  rq_init_comm_if_connected(9, "1")
  rq_init_comm_if_connected(2, "2")
  rq_init_comm_if_connected(3, "3")
  rq_init_comm_if_connected(4, "4")
  rq_print_connected_grippers()
  rq_gripper_communication_thread = run rq_gripper_communication()
  set_closed_norm(100.0, 1)
  set_open_norm(0.0, 1)
  set_closed_mm(0.0, 1)
  set_open_mm(50.0, 1)
  set_closed_norm(100.0, 2)
  set_open_norm(0.0, 2)
  set_closed_mm(0.0, 2)
  set_open_mm(50.0, 2)
  set_closed_norm(100.0, 3)
  set_open_norm(0.0, 3)
  set_closed_mm(0.0, 3)
  set_open_mm(50.0, 3)
  set_closed_norm(100.0, 4)
  set_open_norm(0.0, 4)
  set_closed_mm(0.0, 4)
  set_open_mm(50.0, 4)
  rq_current_limit_enabled = False
  while(not rq_gripper_communication_thread_started):
      sleep(0.008)
  end
  # end: URCap Installation Node
  global Pallet_2_cnt_3=1
  global Pallet_2_cnt_4=1
  global Pallet_2_cnt_5=1
  global Pallet_2_cnt_6=1
  global Pallet_2_lct_3=1
  global Pallet_2_lct_4=1
  global Pallet_2_lct_5=1
  global Pallet_2_lct_6=1
  global Pallet_2_lno_3=1
  global Pallet_2_lno_4=1
  global Pallet_2_lno_5=1
  global Pallet_2_lno_6=1
  global Pallet_2_sep_3= False
  global Pallet_2_sep_4= False
  global Pallet_2_sep_5= False
  global Pallet_2_sep_6= False
  global Pallet_2_tct_3=1
  global Pallet_2_tct_4=1
  global Pallet_2_tct_5=1
  global Pallet_2_tct_6=1
  global qNearApproach=[0,0,0,0,0,0]
  global qNearApproach_1=[0,0,0,0,0,0]
  global qNearApproach_2=[0,0,0,0,0,0]
  global qNearApproach_3=[0,0,0,0,0,0]
  global Waypoint_2_p=p[.497545315671, .066443275206, .565567908320, 2.166165135185, -2.096986285032, -.058830025629]
  global Waypoint_2_q=[3.020538828963275, -1.5350072347942687, 1.310240075700583, -1.2376589337904829, -1.6454681359193124, -0.14796686856282548]
  global Approach_1_p=p[.529811548736, .078794296821, -.249075713058, 2.252782682541, -2.172328817817, .036580928376]
  global Approach_1_q=[3.039864276185085, -0.18566656279727667, 1.7536743022026577, -3.1489013797878584, -1.5954024336410413, -0.13295549283606078]
  global ToolActionPoi_1_p=p[.529805653595, .078793026024, -.279911555553, 2.252768683998, -2.172326347106, .036578768693]
  global ToolActionPoi_1_q=[3.039744912416083, -0.11220692465133553, 1.6920841553070907, -3.16078404588802, -1.5955704096675678, -0.13312653598666024]
  global Exit_2_p=p[.529810238319, .078794594586, -.211983202439, 2.252768831616, -2.172321661670, .036580192861]
  global Exit_2_q=[3.0400074576796485, -0.2750556215204334, 1.820883845919285, -3.1267173172014413, -1.5952202467689496, -0.13278613781927362]
  global Approach_p=p[.259939147756, -.683221746138, .330823595725, .096711987287, 3.097647085282, .045794034220]
  global Approach_q=[1.7433785897016765, -0.9789911612274125, 1.1929114404367116, -1.7636157466916895, -1.5217364879006539, 0.23748448608004402]
  global ToolActionPoint_p=p[.260951127880, -.682556749615, .307415310056, .096720171615, 3.097650623093, .045741938859]
  global ToolActionPoint_q=[1.7448971700273574, -0.9655793386006408, 1.2326464916352902, -1.816818537032935, -1.5217211095327015, 0.23910702792430083]
  global Exit_1_p=p[.258824165549, -.683958688734, .356887144820, .096737432605, 3.097619259377, .045729561599]
  global Exit_1_q=[1.741693917054314, -0.990422118385399, 1.1437541193824776, -1.7029416535283248, -1.5217729231978865, 0.23566896849839264]
  while (True):
    $ 2 "Robot Program"
    $ 3 "Home (Safe)"
    movej([2.5829941725145966, -1.8029425748621035, 2.4397996453919744, -3.810050312281298, -1.0067438250200702, 0.02806297247002032], a=1.3962634015954636, v=1.0471975511965976)
    # begin: URCap Program Node
    #   Source: EnabledRobotics - ER-ABILITY, 5.0.0, Enabled Robotics ApS
    #   Type: ER-Ability
    $ 4 "ER-Ability"
    __er_thread_handle = 0
    daemon=rpc_factory("xmlrpc", "http://192.168.11.40:4568")
    daemon.set_init_status(0)
    HOST_IP = ""
    interpreter_mode(clearQueueOnEnter=False, clearOnEnd=False)
    if (not daemon.connect(HOST_IP)):
      textmsg("Failed to connect to ability")
      halt
    end
    thread __er_connection_watchdog():
      while (True):
        if (not daemon.watchdog()):
          textmsg("Lost connection to ability")
          halt
        end
        sleep(3.0)
      end
    end
    def sendError(errorMsg):
    daemon.send_error(errorMsg)
  end
  daemon.set_init_status(1)
  __er_watchdog_handle = run __er_connection_watchdog()
  interpreter_mode(clearQueueOnEnter=False, clearOnEnd=False)
  # begin: URCap Program Node
  #   Source: EnabledRobotics - ER-ABILITY, 5.0.0, Enabled Robotics ApS
  #   Type: EventNode
  $ 5 "EventNode: GripOpen" "noBreak"
  def GripOpen_definition():
  # begin: URCap Program Node
  #   Source: Robotiq_Grippers, 2.4.0.45103, Robotiq Inc.
  #   Type: Gripper
  $ 6 "Gripper Open (1)" "noBreak"
  if not(gripper_connected[0]):
    popup("Gripper 1 must be connected to run this program.", "No connection", False, True, True)
  end
  if not(rq_is_gripper_activated("1")):
    popup("Gripper 1 is not activated. Go to Installation tab > Gripper to activate it and run the program again.", "Not activated", False, True, True)
  end
  rq_set_pos_spd_for(0, 255, 255, "1")
  rq_wait_pos_spe_for_request(0, 255, 255, "1")
  rq_go_to("1")
  rq_wait("1")
  # end: URCap Program Node
  end
  thread GripOpen_thread():
  GripOpen_definition()
  daemon.done_executing()
  end
  def GripOpen():
  textmsg("Executing event: GripOpen")
  __er_thread_handle = run GripOpen_thread()
  end
  if (not daemon.register_method("GripOpen","[]", False)):
    textmsg("Failed to connect to register method GripOpen")
    halt
  end
  sync()
  # end: URCap Program Node
  # begin: URCap Program Node
  #   Source: EnabledRobotics - ER-ABILITY, 5.0.0, Enabled Robotics ApS
  #   Type: EventNode
  $ 7 "EventNode: GripClosed" "noBreak"
  def GripClosed_definition():
  # begin: URCap Program Node
  #   Source: Robotiq_Grippers, 2.4.0.45103, Robotiq Inc.
  #   Type: Gripper
  $ 8 "Gripper Close (1)" "noBreak"
  if not(gripper_connected[0]):
    popup("Gripper 1 must be connected to run this program.", "No connection", False, True, True)
  end
  if not(rq_is_gripper_activated("1")):
    popup("Gripper 1 is not activated. Go to Installation tab > Gripper to activate it and run the program again.", "Not activated", False, True, True)
  end
  rq_set_pos_spd_for(255, 255, 179, "1")
  rq_wait_pos_spe_for_request(255, 255, 179, "1")
  rq_go_to("1")
  rq_wait("1")
  # end: URCap Program Node
  end
  thread GripClosed_thread():
  GripClosed_definition()
  daemon.done_executing()
  end
  def GripClosed():
  textmsg("Executing event: GripClosed")
  __er_thread_handle = run GripClosed_thread()
  end
  if (not daemon.register_method("GripClosed","[]", False)):
    textmsg("Failed to connect to register method GripClosed")
    halt
  end
  sync()
  # end: URCap Program Node
  # begin: URCap Program Node
  #   Source: EnabledRobotics - ER-ABILITY, 5.0.0, Enabled Robotics ApS
  #   Type: EventNode
  $ 9 "EventNode: Unload" "noBreak"
  global __er_Unload_arg_pose = p[0, 0, 0, 0, 0, 0]
  def Unload_definition(arg_pose):
  $ 10 "Unload_ref≔__er_Unload_arg_pose" "noBreak"
  global Unload_ref=__er_Unload_arg_pose
  $ 11 "MoveJ" "noBreak"
  $ 12 "Waypoint_2" "noBreak"
  movej(get_inverse_kin(Waypoint_2_p, qnear=Waypoint_2_q), a=1.3962634015954636, v=1.0471975511965976)
  $ 13 "Pallet_5" "noBreak"
  def Pallet_5_trans(pose):
  return p[pose[0], pose[1], pose[2], 0, 0, 0]
  end
  def Pallet_5_rot(pose):
  return p[0, 0, 0, pose[3], pose[4], pose[5]]
  end
  def Pallet_5_compute_pallet_waypoint(T_base_feature_taught, T_feature_referencePoint_taught, T_referencePoint_approach_taught, T_base_feature, T_base_referencePoint):
  local trans_referencePoint_approach_in_feature_taught = pose_sub(Pallet_5_trans(pose_trans(T_feature_referencePoint_taught, T_referencePoint_approach_taught)), Pallet_5_trans(T_feature_referencePoint_taught))
  local rot_referencePoint_approach_in_feature_taught = pose_trans(Pallet_5_rot(T_feature_referencePoint_taught), pose_trans(Pallet_5_rot(T_referencePoint_approach_taught), pose_inv(Pallet_5_rot(T_feature_referencePoint_taught))))
  T_feature_referencePoint = pose_trans(pose_inv(T_base_feature), T_base_referencePoint)
  rot_referencePoint_approach = pose_trans(pose_inv(Pallet_5_rot(T_feature_referencePoint)), pose_trans(rot_referencePoint_approach_in_feature_taught, Pallet_5_rot(T_feature_referencePoint)))
  T_feature_approach = pose_trans(trans_referencePoint_approach_in_feature_taught, pose_trans(T_feature_referencePoint, rot_referencePoint_approach))
  T_base_approach = pose_trans(T_base_feature, T_feature_approach)
  return T_base_approach
  end
  Pallet_2_tct_6 = 3
  if (Pallet_2_cnt_6 > 3 or Pallet_2_cnt_6 < 1):
    Pallet_2_cnt_6 = 1
  end
  $ 14 "Patterns" "noBreak"
  $ 15 "Line_Pattern_7" "noBreak"
  $ 18 "Layers" "noBreak"
  if (Pallet_2_cnt_6 < 4):
    Pallet_2_lno_6 = 1
    Pallet_2_lct_6 = Pallet_2_cnt_6
    global StartItem_7=pose_trans(p[0.0,0.0,0.0,0.0,0.0,0.0], pose_trans(p[-.000000000000, -.000000000000, -.000000000000, .000000000000, .000000000000, .000000000000], p[.529805653595, .078793026024, -.279911555553, 2.252768683999, -2.172326347101, .036578768700]))
    global EndItem_7=pose_trans(p[0.0,0.0,0.0,0.0,0.0,0.0], pose_trans(p[-.000000000000, -.000000000000, -.000000000000, .000000000000, .000000000000, .000000000000], p[.533401069223, -.101391020004, -.279793718806, 2.252783599118, -2.172333887579, .036654201565]))
    referencePoin_1 = interpolate_pose(StartItem_7, EndItem_7, (Pallet_2_lct_6 - 1)/2)
    if ((Pallet_2_lct_6 - 1) < 1.5):
      qNearApproach_1 = [2.885448189355559, 0.43603101886187573, 1.512248322517327, -5.09598803422031, -1.2812075252986297, -0.023929430846770572]
    else:
      qNearApproach_1 = [2.272042773983432, 0.4199865702204392, 1.4836778687882308, -5.05440269585694, -0.667839702259915, -0.018231839794984772]
    end
    direction = p[0,0,1,0,0,0]
    referencePoin_1 = pose_add (referencePoin_1,p[0.0*direction[0],0.0*direction[1],0.0*direction[2],0,0,0])
  end
  Approach_1_p = Pallet_5_compute_pallet_waypoint(p[0.0,0.0,0.0,0.0,0.0,0.0], pose_trans(pose_inv(p[0.0,0.0,0.0,0.0,0.0,0.0]), p[0.5298056535954119,0.07879302602441744,-0.279911555552729,2.2527686839987453,-2.1723263471008782,0.03657876870047535]), p[7.713003808866858E-4,-2.4326214461312112E-4,-0.030825235408129148,9.465437041250408E-6,-7.291023033565463E-6,-4.926570927565642E-6], p[0.0,0.0,0.0,0.0,0.0,0.0], referencePoin_1)
  Approach_1_p = pose_trans(p[0.5298056535954119,0.07879302602441744,-0.279911555552729,2.252768683998824,-2.1723263471009577,0.03657876870045813], pose_trans(pose_inv(referencePoin_1), Approach_1_p))
  Approach_1_q = qNearApproach_1
  ToolActionPoi_1_p = Pallet_5_compute_pallet_waypoint(p[0.0,0.0,0.0,0.0,0.0,0.0], pose_trans(pose_inv(p[0.0,0.0,0.0,0.0,0.0,0.0]), p[0.5298056535954119,0.07879302602441744,-0.279911555552729,2.2527686839987453,-2.1723263471008782,0.03657876870047535]), p[1.3877787807814457E-17,0.0,0.0,0.0,0.0,0.0], p[0.0,0.0,0.0,0.0,0.0,0.0], referencePoin_1)
  ToolActionPoi_1_p = pose_trans(p[0.5298056535954119,0.07879302602441744,-0.279911555552729,2.252768683998824,-2.1723263471009577,0.03657876870045813], pose_trans(pose_inv(referencePoin_1), ToolActionPoi_1_p))
  Exit_2_p = Pallet_5_compute_pallet_waypoint(p[0.0,0.0,0.0,0.0,0.0,0.0], pose_trans(pose_inv(p[0.0,0.0,0.0,0.0,0.0,0.0]), p[0.5298056535954119,0.07879302602441744,-0.279911555552729,2.2527686839987453,-2.1723263471008782,0.03657876870047535]), p[0.0017000247291813209,-5.274420544957303E-4,-0.06790502854043742,-1.5766278052156214E-6,2.8353740061571936E-6,-2.251562946520516E-6], p[0.0,0.0,0.0,0.0,0.0,0.0], referencePoin_1)
  Exit_2_p = pose_trans(p[0.5298056535954119,0.07879302602441744,-0.279911555552729,2.252768683998824,-2.1723263471009577,0.03657876870045813], pose_trans(pose_inv(referencePoin_1), Exit_2_p))
  $ 19 "At Each Item" "noBreak"
  $ 20 "Generated Movements" "noBreak"
  $ 21 "MoveJ" "noBreak"
  $ 22 "Approach_1" "noBreak"
  movej(get_inverse_kin(pose_trans(referencePoin_1, pose_trans(p[.066528706245, .530155020651, -.282422442075, -2.252768683999, 2.172326347101, -.036578768700], Approach_1_p)), qnear=Approach_1_q), a=1.3962634015954636, v=1.0471975511965976)
  $ 23 "MoveL" "noBreak"
  $ 24 "ToolActionPoi_1" "noBreak"
  movel(pose_trans(referencePoin_1, pose_trans(p[.066528706245, .530155020651, -.282422442075, -2.252768683999, 2.172326347101, -.036578768700], ToolActionPoi_1_p)), a=1.2, v=0.25)
  $ 25 "Tool action" "noBreak"
  # begin: URCap Program Node
  #   Source: Robotiq_Grippers, 2.4.0.45103, Robotiq Inc.
  #   Type: Gripper
  $ 26 "Gripper Close (1)" "noBreak"
  if not(gripper_connected[0]):
    popup("Gripper 1 must be connected to run this program.", "No connection", False, True, True)
  end
  if not(rq_is_gripper_activated("1")):
    popup("Gripper 1 is not activated. Go to Installation tab > Gripper to activate it and run the program again.", "Not activated", False, True, True)
  end
  rq_set_pos_spd_for(255, 255, 255, "1")
  rq_wait_pos_spe_for_request(255, 255, 255, "1")
  rq_go_to("1")
  rq_wait("1")
  # end: URCap Program Node
  $ 27 "MoveL" "noBreak"
  $ 28 "Exit_2" "noBreak"
  movel(pose_trans(referencePoin_1, pose_trans(p[.066528706245, .530155020651, -.282422442075, -2.252768683999, 2.172326347101, -.036578768700], Exit_2_p)), a=1.2, v=0.25)
  Pallet_2_sep_6 = False
  if (Pallet_2_cnt_6 >= 3):
    Pallet_2_cnt_6 = 1
  else:
    Pallet_2_cnt_6 = Pallet_2_cnt_6 + 1
  end
  $ 29 "MoveJ" "noBreak"
  $ 30 "Waypoint_2" "noBreak"
  movej(get_inverse_kin(Waypoint_2_p, qnear=Waypoint_2_q), a=1.3962634015954636, v=1.0471975511965976)
  $ 31 "Pallet_1" "noBreak"
  def Pallet_1_trans(pose):
  return p[pose[0], pose[1], pose[2], 0, 0, 0]
  end
  def Pallet_1_rot(pose):
  return p[0, 0, 0, pose[3], pose[4], pose[5]]
  end
  def Pallet_1_compute_pallet_waypoint(T_base_feature_taught, T_feature_referencePoint_taught, T_referencePoint_approach_taught, T_base_feature, T_base_referencePoint):
  local trans_referencePoint_approach_in_feature_taught = pose_sub(Pallet_1_trans(pose_trans(T_feature_referencePoint_taught, T_referencePoint_approach_taught)), Pallet_1_trans(T_feature_referencePoint_taught))
  local rot_referencePoint_approach_in_feature_taught = pose_trans(Pallet_1_rot(T_feature_referencePoint_taught), pose_trans(Pallet_1_rot(T_referencePoint_approach_taught), pose_inv(Pallet_1_rot(T_feature_referencePoint_taught))))
  T_feature_referencePoint = pose_trans(pose_inv(T_base_feature), T_base_referencePoint)
  rot_referencePoint_approach = pose_trans(pose_inv(Pallet_1_rot(T_feature_referencePoint)), pose_trans(rot_referencePoint_approach_in_feature_taught, Pallet_1_rot(T_feature_referencePoint)))
  T_feature_approach = pose_trans(trans_referencePoint_approach_in_feature_taught, pose_trans(T_feature_referencePoint, rot_referencePoint_approach))
  T_base_approach = pose_trans(T_base_feature, T_feature_approach)
  return T_base_approach
  end
  Pallet_2_tct_5 = 3
  if (Pallet_2_cnt_5 > 3 or Pallet_2_cnt_5 < 1):
    Pallet_2_cnt_5 = 1
  end
  $ 32 "Patterns" "noBreak"
  $ 33 "Line_Pattern_1" "noBreak"
  $ 36 "Layers" "noBreak"
  if (Pallet_2_cnt_5 < 4):
    Pallet_2_lno_5 = 1
    Pallet_2_lct_5 = Pallet_2_cnt_5
    global StartItem_1=pose_trans(Unload_ref, pose_trans(p[.418279672309, .619551005398, .340218691369, -.096685752657, -3.097655012832, -.045744274097], p[.260951127880, -.682556749615, .307415310056, .096720171636, 3.097650623082, .045741938829]))
    global EndItem_1=pose_trans(Unload_ref, pose_trans(p[.418279672309, .619551005398, .340218691369, -.096685752657, -3.097655012832, -.045744274097], p[.082322324479, -.670818754149, .307468197109, .096703817876, 3.097665036034, .045785718306]))
    referencePoin_2 = interpolate_pose(StartItem_1, EndItem_1, (Pallet_2_lct_5 - 1)/2)
    if ((Pallet_2_lct_5 - 1) < 1.5):
      qNearApproach_2 = [3.3641552695356225, -0.8479015660023324, 1.98966712800588, -1.131219804936615, -2.916013250302344, 0.010451340576699941]
    else:
      qNearApproach_2 = [3.300396662600974, -0.612779437790441, 1.4440990949301122, -0.8163897168853449, -2.98016670938038, 0.01484693428962075]
    end
    direction = pose_trans(p[0,0,0,Unload_ref[3],Unload_ref[4],Unload_ref[5]], p[0,0,1,0,0,0])
    referencePoin_2 = pose_add (referencePoin_2,p[0.0*direction[0],0.0*direction[1],0.0*direction[2],0,0,0])
  end
  Approach_p = Pallet_1_compute_pallet_waypoint(p[0.3642472151847146,-0.6539896130686794,0.3378929456834839,0.09668575265698816,3.0976550128318143,0.04574427409651193], pose_trans(pose_inv(p[0.3642472151847146,-0.6539896130686794,0.3378929456834839,0.09668575265698816,3.0976550128318143,0.04574427409651193]), p[0.260951127880279,-0.6825567496145907,0.307415310056378,0.09672017163594536,3.0976506230824565,0.04574193882899084]), p[4.300908552967719E-6,-4.9422491205097785E-6,-0.023439584449423678,-3.3818317637974754E-5,-1.900639287119668E-6,-4.541078724455231E-6], Unload_ref, referencePoin_2)
  Approach_p = pose_trans(p[0.2609511278802791,-0.6825567496145908,0.30741531005637773,0.0967201716359448,3.0976506230824357,0.04574193882899086], pose_trans(pose_inv(referencePoin_2), Approach_p))
  Approach_q = qNearApproach_2
  ToolActionPoint_p = Pallet_1_compute_pallet_waypoint(p[0.3642472151847146,-0.6539896130686794,0.3378929456834839,0.09668575265698816,3.0976550128318143,0.04574427409651193], pose_trans(pose_inv(p[0.3642472151847146,-0.6539896130686794,0.3378929456834839,0.09668575265698816,3.0976550128318143,0.04574427409651193]), p[0.260951127880279,-0.6825567496145907,0.307415310056378,0.09672017163594536,3.0976506230824565,0.04574193882899084]), p[5.551115123125783E-17,1.1102230246251565E-16,-3.3306690738754696E-16,0.0,0.0,0.0], Unload_ref, referencePoin_2)
  ToolActionPoint_p = pose_trans(p[0.2609511278802791,-0.6825567496145908,0.30741531005637773,0.0967201716359448,3.0976506230824357,0.04574193882899086], pose_trans(pose_inv(referencePoin_2), ToolActionPoint_p))
  Exit_1_p = Pallet_1_compute_pallet_waypoint(p[0.3642472151847146,-0.6539896130686794,0.3378929456834839,0.09668575265698816,3.0976550128318143,0.04574427409651193], pose_trans(pose_inv(p[0.3642472151847146,-0.6539896130686794,0.3378929456834839,0.09668575265698816,3.0976550128318143,0.04574427409651193]), p[0.260951127880279,-0.6825567496145907,0.307415310056378,0.09672017163594536,3.0976506230824565,0.04574193882899084]), p[-2.4468940774680092E-6,-6.239484140468932E-6,-0.04953737772677924,6.96031944656997E-6,-3.138925438944591E-5,1.1138535086107724E-5], Unload_ref, referencePoin_2)
  Exit_1_p = pose_trans(p[0.2609511278802791,-0.6825567496145908,0.30741531005637773,0.0967201716359448,3.0976506230824357,0.04574193882899086], pose_trans(pose_inv(referencePoin_2), Exit_1_p))
  $ 37 "At Each Item" "noBreak"
  $ 38 "Generated Movements" "noBreak"
  $ 39 "MoveJ" "noBreak"
  $ 40 "Approach" "noBreak"
  movej(get_inverse_kin(pose_trans(referencePoin_2, pose_trans(p[.315836214354, .655355973761, .315022878219, -.096720171636, -3.097650623082, -.045741938829], Approach_p)), qnear=Approach_q), a=1.3962634015954636, v=1.0471975511965976)
  $ 41 "MoveL" "noBreak"
  $ 42 "ToolActionPoint" "noBreak"
  movel(pose_trans(referencePoin_2, pose_trans(p[.315836214354, .655355973761, .315022878219, -.096720171636, -3.097650623082, -.045741938829], ToolActionPoint_p)), a=1.2, v=0.25)
  $ 43 "Tool action" "noBreak"
  # begin: URCap Program Node
  #   Source: Robotiq_Grippers, 2.4.0.45103, Robotiq Inc.
  #   Type: Gripper
  $ 44 "Gripper Open (1)" "noBreak"
  if not(gripper_connected[0]):
    popup("Gripper 1 must be connected to run this program.", "No connection", False, True, True)
  end
  if not(rq_is_gripper_activated("1")):
    popup("Gripper 1 is not activated. Go to Installation tab > Gripper to activate it and run the program again.", "Not activated", False, True, True)
  end
  rq_set_pos_spd_for(0, 255, 255, "1")
  rq_wait_pos_spe_for_request(0, 255, 255, "1")
  rq_go_to("1")
  rq_wait("1")
  # end: URCap Program Node
  $ 45 "MoveL" "noBreak"
  $ 46 "Exit_1" "noBreak"
  movel(pose_trans(referencePoin_2, pose_trans(p[.315836214354, .655355973761, .315022878219, -.096720171636, -3.097650623082, -.045741938829], Exit_1_p)), a=1.2, v=0.25)
  Pallet_2_sep_5 = False
  if (Pallet_2_cnt_5 >= 3):
    Pallet_2_cnt_5 = 1
  else:
    Pallet_2_cnt_5 = Pallet_2_cnt_5 + 1
  end
  $ 47 "MoveJ" "noBreak"
  $ 48 "Waypoint_2" "noBreak"
  movej(get_inverse_kin(Waypoint_2_p, qnear=Waypoint_2_q), a=1.3962634015954636, v=1.0471975511965976)
  end
  thread Unload_thread():
  Unload_definition(__er_Unload_arg_pose)
  daemon.done_executing()
  end
  def Unload(arg_pose):
  textmsg("Executing event: Unload, with arguments:")
  textmsg("Argument: arg_pose = ", arg_pose)
  __er_Unload_arg_pose = arg_pose
  __er_thread_handle = run Unload_thread()
  end
  if (not daemon.register_method("Unload","[pose]", False)):
    textmsg("Failed to connect to register method Unload")
    halt
  end
  sync()
  # end: URCap Program Node
  # begin: URCap Program Node
  #   Source: EnabledRobotics - ER-ABILITY, 5.0.0, Enabled Robotics ApS
  #   Type: EventNode
  $ 49 "EventNode: Palletize" "noBreak"
  global __er_Palletize_arg_pose = p[0, 0, 0, 0, 0, 0]
  def Palletize_definition(arg_pose):
  $ 50 "Pallet_ref≔__er_Palletize_arg_pose" "noBreak"
  global Pallet_ref=__er_Palletize_arg_pose
  $ 51 "MoveJ" "noBreak"
  $ 52 "Waypoint_2" "noBreak"
  movej(get_inverse_kin(Waypoint_2_p, qnear=Waypoint_2_q), a=1.3962634015954636, v=1.0471975511965976)
  $ 53 "Pallet_3" "noBreak"
  def Pallet_3_trans(pose):
  return p[pose[0], pose[1], pose[2], 0, 0, 0]
  end
  def Pallet_3_rot(pose):
  return p[0, 0, 0, pose[3], pose[4], pose[5]]
  end
  def Pallet_3_compute_pallet_waypoint(T_base_feature_taught, T_feature_referencePoint_taught, T_referencePoint_approach_taught, T_base_feature, T_base_referencePoint):
  local trans_referencePoint_approach_in_feature_taught = pose_sub(Pallet_3_trans(pose_trans(T_feature_referencePoint_taught, T_referencePoint_approach_taught)), Pallet_3_trans(T_feature_referencePoint_taught))
  local rot_referencePoint_approach_in_feature_taught = pose_trans(Pallet_3_rot(T_feature_referencePoint_taught), pose_trans(Pallet_3_rot(T_referencePoint_approach_taught), pose_inv(Pallet_3_rot(T_feature_referencePoint_taught))))
  T_feature_referencePoint = pose_trans(pose_inv(T_base_feature), T_base_referencePoint)
  rot_referencePoint_approach = pose_trans(pose_inv(Pallet_3_rot(T_feature_referencePoint)), pose_trans(rot_referencePoint_approach_in_feature_taught, Pallet_3_rot(T_feature_referencePoint)))
  T_feature_approach = pose_trans(trans_referencePoint_approach_in_feature_taught, pose_trans(T_feature_referencePoint, rot_referencePoint_approach))
  T_base_approach = pose_trans(T_base_feature, T_feature_approach)
  return T_base_approach
  end
  Pallet_2_tct_3 = 3
  if (Pallet_2_cnt_3 > 3 or Pallet_2_cnt_3 < 1):
    Pallet_2_cnt_3 = 1
  end
  $ 54 "Patterns" "noBreak"
  $ 55 "Line_Pattern_5" "noBreak"
  $ 58 "Layers" "noBreak"
  if (Pallet_2_cnt_3 < 4):
    Pallet_2_lno_3 = 1
    Pallet_2_lct_3 = Pallet_2_cnt_3
    global StartItem_5=pose_trans(Pallet_ref, pose_trans(p[.418279672309, .619551005398, .340218691369, -.096685752657, -3.097655012832, -.045744274097], p[.260951127880, -.682556749615, .307415310056, .096720171636, 3.097650623082, .045741938829]))
    global EndItem_5=pose_trans(Pallet_ref, pose_trans(p[.418279672309, .619551005398, .340218691369, -.096685752657, -3.097655012832, -.045744274097], p[.082322324479, -.670818754149, .307468197109, .096703817876, 3.097665036034, .045785718306]))
    referencePoin_3 = interpolate_pose(StartItem_5, EndItem_5, (Pallet_2_lct_3 - 1)/2)
    if ((Pallet_2_lct_3 - 1) < 1.5):
      qNearApproach = [1.8853350729711007, -0.9945419025980371, 1.8756705078246672, -3.9864826836818184, -1.9494013418490388, 0.0576506840721043]
    else:
      qNearApproach = [1.4834301388931141, -1.1270563789595887, 2.126921432265375, -4.109054351196034, -1.5477728899200969, 0.04377366676978213]
    end
    direction = pose_trans(p[0,0,0,Pallet_ref[3],Pallet_ref[4],Pallet_ref[5]], p[0,0,1,0,0,0])
    referencePoin_3 = pose_add (referencePoin_3,p[0.0*direction[0],0.0*direction[1],0.0*direction[2],0,0,0])
  end
  Approach_p = Pallet_3_compute_pallet_waypoint(p[0.3642472151847146,-0.6539896130686794,0.3378929456834839,0.09668575265698816,3.0976550128318143,0.04574427409651193], pose_trans(pose_inv(p[0.3642472151847146,-0.6539896130686794,0.3378929456834839,0.09668575265698816,3.0976550128318143,0.04574427409651193]), p[0.260951127880279,-0.6825567496145907,0.307415310056378,0.09672017163594536,3.0976506230824565,0.04574193882899084]), p[4.300908552967719E-6,-4.9422491205097785E-6,-0.023439584449423678,-3.3818317637974754E-5,-1.900639287119668E-6,-4.541078724455231E-6], Pallet_ref, referencePoin_3)
  Approach_p = pose_trans(p[0.2609511278802791,-0.6825567496145908,0.30741531005637773,0.0967201716359448,3.0976506230824357,0.04574193882899086], pose_trans(pose_inv(referencePoin_3), Approach_p))
  Approach_q = qNearApproach
  ToolActionPoint_p = Pallet_3_compute_pallet_waypoint(p[0.3642472151847146,-0.6539896130686794,0.3378929456834839,0.09668575265698816,3.0976550128318143,0.04574427409651193], pose_trans(pose_inv(p[0.3642472151847146,-0.6539896130686794,0.3378929456834839,0.09668575265698816,3.0976550128318143,0.04574427409651193]), p[0.260951127880279,-0.6825567496145907,0.307415310056378,0.09672017163594536,3.0976506230824565,0.04574193882899084]), p[5.551115123125783E-17,1.1102230246251565E-16,-3.3306690738754696E-16,0.0,0.0,0.0], Pallet_ref, referencePoin_3)
  ToolActionPoint_p = pose_trans(p[0.2609511278802791,-0.6825567496145908,0.30741531005637773,0.0967201716359448,3.0976506230824357,0.04574193882899086], pose_trans(pose_inv(referencePoin_3), ToolActionPoint_p))
  Exit_1_p = Pallet_3_compute_pallet_waypoint(p[0.3642472151847146,-0.6539896130686794,0.3378929456834839,0.09668575265698816,3.0976550128318143,0.04574427409651193], pose_trans(pose_inv(p[0.3642472151847146,-0.6539896130686794,0.3378929456834839,0.09668575265698816,3.0976550128318143,0.04574427409651193]), p[0.260951127880279,-0.6825567496145907,0.307415310056378,0.09672017163594536,3.0976506230824565,0.04574193882899084]), p[-2.4468940774680092E-6,-6.239484140468932E-6,-0.04953737772677924,6.96031944656997E-6,-3.138925438944591E-5,1.1138535086107724E-5], Pallet_ref, referencePoin_3)
  Exit_1_p = pose_trans(p[0.2609511278802791,-0.6825567496145908,0.30741531005637773,0.0967201716359448,3.0976506230824357,0.04574193882899086], pose_trans(pose_inv(referencePoin_3), Exit_1_p))
  $ 59 "At Each Item" "noBreak"
  $ 60 "Generated Movements" "noBreak"
  $ 61 "MoveJ" "noBreak"
  $ 62 "Approach" "noBreak"
  set_tcp(p[0.0,0.0,0.0,0.0,0.0,0.0])
  movej(get_inverse_kin(pose_trans(referencePoin_3, pose_trans(p[.315836214354, .655355973761, .315022878219, -.096720171636, -3.097650623082, -.045741938829], Approach_p)), qnear=Approach_q), a=1.3962634015954636, v=1.0471975511965976)
  $ 63 "MoveL" "noBreak"
  $ 64 "ToolActionPoint" "noBreak"
  movel(pose_trans(referencePoin_3, pose_trans(p[.315836214354, .655355973761, .315022878219, -.096720171636, -3.097650623082, -.045741938829], ToolActionPoint_p)), a=1.2, v=0.25)
  $ 65 "Tool action" "noBreak"
  # begin: URCap Program Node
  #   Source: Robotiq_Grippers, 2.4.0.45103, Robotiq Inc.
  #   Type: Gripper
  $ 66 "Gripper Close (1)" "noBreak"
  if not(gripper_connected[0]):
    popup("Gripper 1 must be connected to run this program.", "No connection", False, True, True)
  end
  if not(rq_is_gripper_activated("1")):
    popup("Gripper 1 is not activated. Go to Installation tab > Gripper to activate it and run the program again.", "Not activated", False, True, True)
  end
  rq_set_pos_spd_for(255, 250, 0, "1")
  rq_wait_pos_spe_for_request(255, 250, 0, "1")
  rq_go_to("1")
  rq_wait("1")
  # end: URCap Program Node
  $ 67 "MoveL" "noBreak"
  $ 68 "Exit_1" "noBreak"
  movel(pose_trans(referencePoin_3, pose_trans(p[.315836214354, .655355973761, .315022878219, -.096720171636, -3.097650623082, -.045741938829], Exit_1_p)), a=1.2, v=0.25)
  Pallet_2_sep_3 = False
  if (Pallet_2_cnt_3 >= 3):
    Pallet_2_cnt_3 = 1
  else:
    Pallet_2_cnt_3 = Pallet_2_cnt_3 + 1
  end
  $ 69 "MoveJ" "noBreak"
  $ 70 "Waypoint_2" "noBreak"
  movej(get_inverse_kin(Waypoint_2_p, qnear=Waypoint_2_q), a=1.3962634015954636, v=1.0471975511965976)
  $ 71 "Pallet_4" "noBreak"
  def Pallet_4_trans(pose):
  return p[pose[0], pose[1], pose[2], 0, 0, 0]
  end
  def Pallet_4_rot(pose):
  return p[0, 0, 0, pose[3], pose[4], pose[5]]
  end
  def Pallet_4_compute_pallet_waypoint(T_base_feature_taught, T_feature_referencePoint_taught, T_referencePoint_approach_taught, T_base_feature, T_base_referencePoint):
  local trans_referencePoint_approach_in_feature_taught = pose_sub(Pallet_4_trans(pose_trans(T_feature_referencePoint_taught, T_referencePoint_approach_taught)), Pallet_4_trans(T_feature_referencePoint_taught))
  local rot_referencePoint_approach_in_feature_taught = pose_trans(Pallet_4_rot(T_feature_referencePoint_taught), pose_trans(Pallet_4_rot(T_referencePoint_approach_taught), pose_inv(Pallet_4_rot(T_feature_referencePoint_taught))))
  T_feature_referencePoint = pose_trans(pose_inv(T_base_feature), T_base_referencePoint)
  rot_referencePoint_approach = pose_trans(pose_inv(Pallet_4_rot(T_feature_referencePoint)), pose_trans(rot_referencePoint_approach_in_feature_taught, Pallet_4_rot(T_feature_referencePoint)))
  T_feature_approach = pose_trans(trans_referencePoint_approach_in_feature_taught, pose_trans(T_feature_referencePoint, rot_referencePoint_approach))
  T_base_approach = pose_trans(T_base_feature, T_feature_approach)
  return T_base_approach
  end
  Pallet_2_tct_4 = 3
  if (Pallet_2_cnt_4 > 3 or Pallet_2_cnt_4 < 1):
    Pallet_2_cnt_4 = 1
  end
  $ 72 "Patterns" "noBreak"
  $ 73 "Line_Pattern_6" "noBreak"
  $ 76 "Layers" "noBreak"
  if (Pallet_2_cnt_4 < 4):
    Pallet_2_lno_4 = 1
    Pallet_2_lct_4 = Pallet_2_cnt_4
    global StartItem_6=pose_trans(p[0.0,0.0,0.0,0.0,0.0,0.0], pose_trans(p[-.000000000000, -.000000000000, -.000000000000, .000000000000, .000000000000, .000000000000], p[.529805653595, .078793026024, -.279911555553, 2.252768683999, -2.172326347101, .036578768700]))
    global EndItem_6=pose_trans(p[0.0,0.0,0.0,0.0,0.0,0.0], pose_trans(p[-.000000000000, -.000000000000, -.000000000000, .000000000000, .000000000000, .000000000000], p[.533401069223, -.101391020004, -.279793718806, 2.252783599118, -2.172333887579, .036654201565]))
    referencePoin_4 = interpolate_pose(StartItem_6, EndItem_6, (Pallet_2_lct_4 - 1)/2)
    if ((Pallet_2_lct_4 - 1) < 1.5):
      qNearApproach_3 = [2.885448189355559, 0.43603101886187573, 1.512248322517327, -5.09598803422031, -1.2812075252986297, -0.023929430846770572]
    else:
      qNearApproach_3 = [2.272042773983432, 0.4199865702204392, 1.4836778687882308, -5.05440269585694, -0.667839702259915, -0.018231839794984772]
    end
    direction = p[0,0,1,0,0,0]
    referencePoin_4 = pose_add (referencePoin_4,p[0.0*direction[0],0.0*direction[1],0.0*direction[2],0,0,0])
  end
  Approach_1_p = Pallet_4_compute_pallet_waypoint(p[0.0,0.0,0.0,0.0,0.0,0.0], pose_trans(pose_inv(p[0.0,0.0,0.0,0.0,0.0,0.0]), p[0.5298056535954119,0.07879302602441744,-0.279911555552729,2.2527686839987453,-2.1723263471008782,0.03657876870047535]), p[7.713003808866858E-4,-2.4326214461312112E-4,-0.030825235408129148,9.465437041250408E-6,-7.291023033565463E-6,-4.926570927565642E-6], p[0.0,0.0,0.0,0.0,0.0,0.0], referencePoin_4)
  Approach_1_p = pose_trans(p[0.5298056535954119,0.07879302602441744,-0.279911555552729,2.252768683998824,-2.1723263471009577,0.03657876870045813], pose_trans(pose_inv(referencePoin_4), Approach_1_p))
  Approach_1_q = qNearApproach_3
  ToolActionPoi_1_p = Pallet_4_compute_pallet_waypoint(p[0.0,0.0,0.0,0.0,0.0,0.0], pose_trans(pose_inv(p[0.0,0.0,0.0,0.0,0.0,0.0]), p[0.5298056535954119,0.07879302602441744,-0.279911555552729,2.2527686839987453,-2.1723263471008782,0.03657876870047535]), p[1.3877787807814457E-17,0.0,0.0,0.0,0.0,0.0], p[0.0,0.0,0.0,0.0,0.0,0.0], referencePoin_4)
  ToolActionPoi_1_p = pose_trans(p[0.5298056535954119,0.07879302602441744,-0.279911555552729,2.252768683998824,-2.1723263471009577,0.03657876870045813], pose_trans(pose_inv(referencePoin_4), ToolActionPoi_1_p))
  Exit_2_p = Pallet_4_compute_pallet_waypoint(p[0.0,0.0,0.0,0.0,0.0,0.0], pose_trans(pose_inv(p[0.0,0.0,0.0,0.0,0.0,0.0]), p[0.5298056535954119,0.07879302602441744,-0.279911555552729,2.2527686839987453,-2.1723263471008782,0.03657876870047535]), p[0.0017000247291813209,-5.274420544957303E-4,-0.06790502854043742,-1.5766278052156214E-6,2.8353740061571936E-6,-2.251562946520516E-6], p[0.0,0.0,0.0,0.0,0.0,0.0], referencePoin_4)
  Exit_2_p = pose_trans(p[0.5298056535954119,0.07879302602441744,-0.279911555552729,2.252768683998824,-2.1723263471009577,0.03657876870045813], pose_trans(pose_inv(referencePoin_4), Exit_2_p))
  $ 77 "At Each Item" "noBreak"
  $ 78 "Generated Movements" "noBreak"
  $ 79 "MoveJ" "noBreak"
  $ 80 "Approach_1" "noBreak"
  movej(get_inverse_kin(pose_trans(referencePoin_4, pose_trans(p[.066528706245, .530155020651, -.282422442075, -2.252768683999, 2.172326347101, -.036578768700], Approach_1_p)), qnear=Approach_1_q), a=1.3962634015954636, v=1.0471975511965976)
  $ 81 "MoveL" "noBreak"
  $ 82 "ToolActionPoi_1" "noBreak"
  movel(pose_trans(referencePoin_4, pose_trans(p[.066528706245, .530155020651, -.282422442075, -2.252768683999, 2.172326347101, -.036578768700], ToolActionPoi_1_p)), a=1.2, v=0.25)
  $ 83 "Tool action" "noBreak"
  # begin: URCap Program Node
  #   Source: Robotiq_Grippers, 2.4.0.45103, Robotiq Inc.
  #   Type: Gripper
  $ 84 "Gripper Open (1)" "noBreak"
  if not(gripper_connected[0]):
    popup("Gripper 1 must be connected to run this program.", "No connection", False, True, True)
  end
  if not(rq_is_gripper_activated("1")):
    popup("Gripper 1 is not activated. Go to Installation tab > Gripper to activate it and run the program again.", "Not activated", False, True, True)
  end
  rq_set_pos_spd_for(0, 250, 0, "1")
  rq_wait_pos_spe_for_request(0, 250, 0, "1")
  rq_go_to("1")
  rq_wait("1")
  # end: URCap Program Node
  $ 85 "MoveL" "noBreak"
  $ 86 "Exit_2" "noBreak"
  movel(pose_trans(referencePoin_4, pose_trans(p[.066528706245, .530155020651, -.282422442075, -2.252768683999, 2.172326347101, -.036578768700], Exit_2_p)), a=1.2, v=0.25)
  Pallet_2_sep_4 = False
  if (Pallet_2_cnt_4 >= 3):
    Pallet_2_cnt_4 = 1
  else:
    Pallet_2_cnt_4 = Pallet_2_cnt_4 + 1
  end
  $ 87 "MoveJ" "noBreak"
  $ 88 "Waypoint_2" "noBreak"
  movej(get_inverse_kin(Waypoint_2_p, qnear=Waypoint_2_q), a=1.3962634015954636, v=1.0471975511965976)
  end
  thread Palletize_thread():
  Palletize_definition(__er_Palletize_arg_pose)
  daemon.done_executing()
  end
  def Palletize(arg_pose):
  textmsg("Executing event: Palletize, with arguments:")
  textmsg("Argument: arg_pose = ", arg_pose)
  __er_Palletize_arg_pose = arg_pose
  __er_thread_handle = run Palletize_thread()
  end
  if (not daemon.register_method("Palletize","[pose]", False)):
    textmsg("Failed to connect to register method Palletize")
    halt
  end
  sync()
  # end: URCap Program Node
  daemon.end_method_registration()
  daemon.set_init_status(2)
  interpreter_mode(clearQueueOnEnter=False)
  # end: URCap Program Node
  end
end
